(* Retentive Timer Off-Delay - implements a timer-off delay that persists if PLC cycle is stopped. 
When the input becomes FALSE after a TRUE, the elapsed time ET will run through until the output Q becomes TRUE. 
*)
FUNCTION_BLOCK FB_RTOF
VAR_INPUT
	IN 	: BOOL; // Starts timer with falling edge, resets timer with rising edge
	PT 	: TIME; // Time to pass, before Q is set
END_VAR
VAR_OUTPUT
	Q 	: BOOL; // is FALSE, PT seconds after IN had a falling edge
	ET 	: TIME; // Elapsed time
END_VAR
VAR
	stPLC_Task_Info 	: ST_PLC_TASK_INFORMATION;
	tAccumulator 		: TIME;
	nLast_Cycle_Count 	: UDINT;
	eState 				: (IDLE, RUN);
END_VAR

LBL_TOP: 
CASE eState OF
	IDLE: 
		IF IN THEN Q := TRUE; tAccumulator := ET := T#0MS; eState := RUN; JMP LBL_TOP; END_IF
	RUN:
		stPLC_Task_Info := F_Get_PLC_Task_Information();
		IF NOT(IN) AND ((nLast_Cycle_Count <> stPLC_Task_Info.CycleCount) OR nLast_Cycle_Count = 0) THEN 
			Q := ET <> PT;
			IF (ET >= PT) THEN Q := FALSE;  eState := IDLE; JMP LBL_TOP; END_IF
			tAccumulator := tAccumulator + stPLC_Task_Info.tCycleTime; 
			ET := LIMIT(T#0MS, THIS^.Lerp(T#0MS, PT, TO_REAL(tAccumulator)/TO_REAL(PT))-stPLC_Task_Info.tCycleTime, PT);
			END_IF
		nLast_Cycle_Count := stPLC_Task_Info.CycleCount;
		IF IN THEN tAccumulator := ET := T#0MS;END_IF
END_CASE

// Linear interpolation (Lerp) - this method interpolates values between 2 time points.
METHOD PRIVATE Lerp : TIME
VAR_INPUT
	tStart 	: TIME := T#0MS; 
	tFinish : TIME;
	fPercentage : REAL; // Value must be between 0 and 1
END_VAR
// Lerp(Start, Finish, Percentage) = Start + (Finish - Start)*Percentage
Lerp := TO_TIME(TO_REAL(tStart) + TO_REAL(tFinish - tStart)*fPercentage);
END_METHOD

END_FUNCTION_BLOCK

(* stored: Version 1.1.0.1, ProductVersion 3.1.4024.4
   POU FB_RTOF: Id {87f5daad-7f7e-490d-952a-93e6f5384134}, SpecialFunc None
   Method Lerp: Id {36a01201-4a8e-4415-91bf-222a16e52a06} *)
